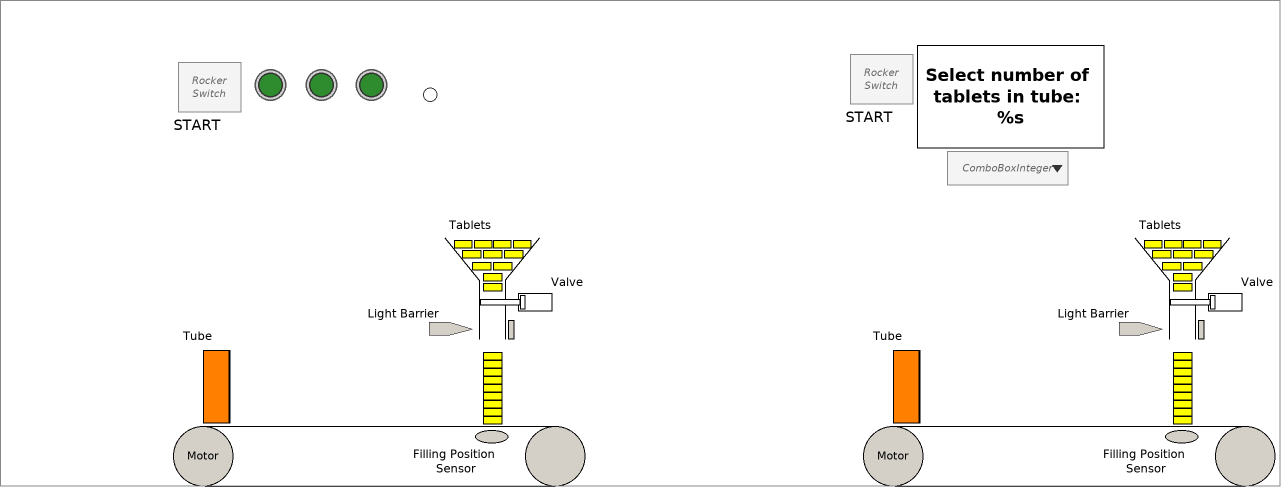
VISUALIZATION Visualization  // 1281x487
    Rectangle (518,293 34x18)
    Rectangle (917,45 187x103), "Select number of tablets in tube: %s", text variable: GVL.TabletsSelected02
    Ellipse (173,426 60x60), "Motor", colour toggle: GVL.MotorRunning01
    Ellipse (525,426 60x60), colour toggle: GVL.MotorRunning01
    Line (205,486) (555,486), colour toggle: GVL.MotorRunning01
    Line (202,426) (555,426), colour toggle: GVL.MotorRunning01
    Label (408,443 96x37), "Filling Position Sensor"
    Rectangle (204,350 26x73)
        p3560616238: Simulation01.TubePosition[1]
    Line (479,280) (479,339)
    Line (505,280) (505,339)
    Line (539,238) (505,280)
    Group (480,295 45x14)
        p3560616238: Simulation01.ValvePosition
        Rectangle (0,4 40x6)
        Rectangle (40,0 5x14)
    Line (479,280) (445,238)
    RoundedRectangle (483,283 19x8)
        p2738717112: Simulation01.TabletPositionVert
    RoundedRectangle (454,240 18x8)
    RoundedRectangle (462,250 19x8)
    RoundedRectangle (472,262 19x8)
    RoundedRectangle (483,273 19x8)
    RoundedRectangle (483,250 19x8)
    RoundedRectangle (493,262 19x8)
    RoundedRectangle (504,250 19x8)
    RoundedRectangle (493,240 18x8)
    RoundedRectangle (474,240 18x8)
    RoundedRectangle (513,240 18x8)
    Ellipse (475,430 33x13), colour toggle: GVL.FillingPosition01
    Label (543,271 48x22), "Valve"
    Label (446,214 48x22), "Tablets"
    Label (171,325 53x22), "Tube"
    Polygon (429,322) (449,322) (472,329) (449,335) (429,335), colour toggle: GVL.LightBarrier01
    Label (355,301 96x25), "Light Barrier"
    Rectangle (508,320 6x19)
    Rectangle (203,350 26x73), invisible if: NOT Simulation01.Tube02Active
        p3560616238: Simulation01.TubePosition[2]
    Rectangle (203,350 26x73), invisible if: NOT Simulation01.Tube03Active
        p3560616238: Simulation01.TubePosition[3]
    RoundedRectangle (483,416 19x8), invisible if: Simulation01.TabletNumberLoaded = 0
        p3560616238: Simulation01.TabletPositionHorizn
    RoundedRectangle (483,408 19x8), invisible if: Simulation01.TabletNumberLoaded < 2
        p3560616238: Simulation01.TabletPositionHorizn
    RoundedRectangle (483,400 19x8), invisible if: Simulation01.TabletNumberLoaded < 3
        p3560616238: Simulation01.TabletPositionHorizn
    RoundedRectangle (483,392 19x8), invisible if: Simulation01.TabletNumberLoaded < 4
        p3560616238: Simulation01.TabletPositionHorizn
    RoundedRectangle (483,384 19x8), invisible if: Simulation01.TabletNumberLoaded < 5
        p3560616238: Simulation01.TabletPositionHorizn
    RoundedRectangle (483,376 19x8), invisible if: Simulation01.TabletNumberLoaded < 6
        p3560616238: Simulation01.TabletPositionHorizn
    RoundedRectangle (483,368 19x8), invisible if: Simulation01.TabletNumberLoaded < 7
        p3560616238: Simulation01.TabletPositionHorizn
    RoundedRectangle (483,360 19x8), invisible if: Simulation01.TabletNumberLoaded < 8
        p3560616238: Simulation01.TabletPositionHorizn
    RoundedRectangle (483,352 19x8), invisible if: Simulation01.TabletNumberLoaded < 9
        p3560616238: Simulation01.TabletPositionHorizn
    Lamp1 (252,64 37x42), variable: GVL.Tablet3Selected01, style: Lamp-Lamp1-Green
    RockerSwitch (178,62 63x50), variable: GVL.StartPb01, behaviour: TOGGLE, style: Switch-RockerSwitch-Blue
    Label (156,114 82x22), "START"
    Lamp1 (303,64 37x42), variable: GVL.Tablet5Selected01, style: Lamp-Lamp1-Green
    Lamp1 (353,64 37x42), variable: GVL.Tablet7Selected01, style: Lamp-Lamp1-Green
    RadioButton (421,41 192x107), variable: Simulation01.VisuTabletsInTube
        Areas[0]: Text=Three tablets in tube
        Areas[1]: Text=Five tablets in tube
        Areas[2]: Text=Seven tablets in tube
    ComboBoxInteger (947,151 121x34), variable: Simulation02.VisuTabletsInTube
    RockerSwitch (850,54 63x50), variable: GVL.StartPb02, behaviour: TOGGLE, style: Switch-RockerSwitch-Blue
    Label (828,106 82x22), "START"
    Rectangle (1208,293 34x18)
    Ellipse (863,426 60x60), "Motor", colour toggle: GVL.MotorRunning02
    Ellipse (1215,426 60x60), colour toggle: GVL.MotorRunning02
    Line (895,486) (1245,486), colour toggle: GVL.MotorRunning02
    Line (892,426) (1245,426), colour toggle: GVL.MotorRunning02
    Label (1098,443 96x37), "Filling Position Sensor"
    Rectangle (894,350 26x73)
        p3560616238: Simulation02.TubePosition[1]
    Line (1169,280) (1169,339)
    Line (1195,280) (1195,339)
    Line (1229,238) (1195,280)
    Group (1170,295 45x14)
        p3560616238: Simulation02.ValvePosition
        Rectangle (0,4 40x6)
        Rectangle (40,0 5x14)
    Line (1169,280) (1135,238)
    RoundedRectangle (1173,283 19x8)
        p2738717112: Simulation02.TabletPositionVert
    RoundedRectangle (1144,240 18x8)
    RoundedRectangle (1152,250 19x8)
    RoundedRectangle (1162,262 19x8)
    RoundedRectangle (1173,273 19x8)
    RoundedRectangle (1173,250 19x8)
    RoundedRectangle (1183,262 19x8)
    RoundedRectangle (1194,250 19x8)
    RoundedRectangle (1183,240 18x8)
    RoundedRectangle (1164,240 18x8)
    RoundedRectangle (1203,240 18x8)
    Ellipse (1165,430 33x13), colour toggle: GVL.FillingPosition02
    Label (1233,271 48x22), "Valve"
    Label (1136,214 48x22), "Tablets"
    Label (861,325 53x22), "Tube"
    Polygon (1119,322) (1139,322) (1162,329) (1139,335) (1119,335), colour toggle: GVL.LightBarrier02
    Label (1045,301 96x25), "Light Barrier"
    Rectangle (1198,320 6x19)
    Rectangle (893,350 26x73), invisible if: NOT Simulation02.Tube02Active
        p3560616238: Simulation02.TubePosition[2]
    Rectangle (893,350 26x73), invisible if: NOT Simulation02.Tube03Active
        p3560616238: Simulation02.TubePosition[3]
    RoundedRectangle (1173,416 19x8), invisible if: Simulation02.TabletNumberLoaded = 0
        p3560616238: Simulation02.TabletPositionHorizn
    RoundedRectangle (1173,408 19x8), invisible if: Simulation02.TabletNumberLoaded < 2
        p3560616238: Simulation02.TabletPositionHorizn
    RoundedRectangle (1173,400 19x8), invisible if: Simulation02.TabletNumberLoaded < 3
        p3560616238: Simulation02.TabletPositionHorizn
    RoundedRectangle (1173,392 19x8), invisible if: Simulation02.TabletNumberLoaded < 4
        p3560616238: Simulation02.TabletPositionHorizn
    RoundedRectangle (1173,384 19x8), invisible if: Simulation02.TabletNumberLoaded < 5
        p3560616238: Simulation02.TabletPositionHorizn
    RoundedRectangle (1173,376 19x8), invisible if: Simulation02.TabletNumberLoaded < 6
        p3560616238: Simulation02.TabletPositionHorizn
    RoundedRectangle (1173,368 19x8), invisible if: Simulation02.TabletNumberLoaded < 7
        p3560616238: Simulation02.TabletPositionHorizn
    RoundedRectangle (1173,360 19x8), invisible if: Simulation02.TabletNumberLoaded < 8
        p3560616238: Simulation02.TabletPositionHorizn
    RoundedRectangle (1173,352 19x8), invisible if: Simulation02.TabletNumberLoaded < 9
        p3560616238: Simulation02.TabletPositionHorizn
END_VISUALIZATION

(* stored: Version 1.1.0.1, ProductVersion 3.1.4024.15
   Visu Visualization: Id {69d51047-4eea-488d-8145-05668e8b9574} *)
